(* IEC 61131-3 sources: Caravan/Archiv/12-04-19/Stations/MachineControl/MachineControl/Class/DayNightSplitter_Class, 1 file *)

(* ---- DayNightSplitter_Class.st ---- *)
(*!
<Class
	Name               = "DayNightSplitter_Class"
	Revision           = "0.0"
	RealtimeTask       = "false"
	CyclicTask         = "true"
	DefCyclictime      = "200 µs"
	BackgroundTask     = "false"
	Sigmatek           = "false"
	OSInterface        = "false"
	HighPriority       = "false"
	Automatic          = "false"
	UpdateMode         = "Prescan"
	SharedCommandTable = "true"
	Objectsize         = "(750,120)">
	<Channels>
		<Server Name="ClassSvr" Visualized="false" Initialize="false" WriteProtected="true" Retentive="false"/>
		<Server Name="DayFanMode" Visualized="true" Initialize="false" WriteProtected="false" Retentive="SRam"/>
		<Server Name="DayFanSpeed" Visualized="true" Initialize="false" WriteProtected="false" Retentive="SRam"/>
		<Server Name="DayHeaterON" Visualized="true" Initialize="false" WriteProtected="false" Retentive="SRam"/>
		<Server Name="DaySetRoomTemp" Visualized="true" Initialize="false" WriteProtected="false" Retentive="SRam"/>
		<Server Name="DaySetTempHZS" Visualized="true" Initialize="false" WriteProtected="false" Retentive="SRam"/>
		<Server Name="NightFanMode" Visualized="true" Initialize="false" WriteProtected="false" Retentive="SRam"/>
		<Server Name="NightFanSpeed" Visualized="true" Initialize="false" WriteProtected="false" Retentive="SRam"/>
		<Server Name="NightHeaterOn" Visualized="true" Initialize="false" WriteProtected="false" Retentive="SRam"/>
		<Server Name="NightSetRoomTemp" Visualized="true" Initialize="false" WriteProtected="false" Retentive="SRam"/>
		<Server Name="NightSetTempHZS" Visualized="true" Initialize="false" WriteProtected="false" Retentive="SRam"/>
		<Client Name="DesiredFanMode" Required="true" Internal="false"/>
		<Client Name="DesiredFanSpeed" Required="true" Internal="false"/>
		<Client Name="DesiredHeaterPWR" Required="true" Internal="false"/>
		<Client Name="DesiredHZSTemp" Required="true" Internal="false"/>
		<Client Name="DesiredRoomTemp" Required="true" Internal="false"/>
		<Client Name="OC_ToTimerClass" Required="true" Internal="false"/>
	</Channels>
</Class>
*)
DayNightSplitter_Class : CLASS
  //Servers:
	ClassSvr 	: SvrChCmd_DINT;
	DaySetTempHZS 	: SvrCh_DINT;
	DaySetRoomTemp 	: SvrCh_DINT;
	DayHeaterON 	: SvrCh_DINT;
	DayFanMode 	: SvrCh_DINT;
	DayFanSpeed 	: SvrCh_DINT;
	NightSetTempHZS 	: SvrCh_DINT;
	NightSetRoomTemp 	: SvrCh_DINT;
	NightHeaterOn 	: SvrCh_DINT;
	NightFanMode 	: SvrCh_DINT;
	NightFanSpeed 	: SvrCh_DINT;
  //Clients:
	OC_ToTimerClass 	: CltChCmd_Timer_Class;
	DesiredHZSTemp 	: CltCh_DINT;
	DesiredRoomTemp 	: CltCh_DINT;
	DesiredHeaterPWR 	: CltCh_DINT;
	DesiredFanMode 	: CltCh_DINT;
	DesiredFanSpeed 	: CltCh_DINT;
  //Variables:
  //Functions:

	FUNCTION VIRTUAL GLOBAL CyWork
		VAR_INPUT
			EAX 	: UDINT;
		END_VAR
		VAR_OUTPUT
			state (EAX) 	: UDINT;
		END_VAR;
  //Tables:
	FUNCTION @STD
		VAR_OUTPUT
			ret_code	: CONFSTATES;
		END_VAR;
	FUNCTION GLOBAL TAB @CT_;
END_CLASS;

#pragma usingLtd Timer_Class

FUNCTION VIRTUAL GLOBAL DayNightSplitter_Class::CyWork
	VAR_INPUT
		EAX 	: UDINT;
	END_VAR
	VAR_OUTPUT
		state (EAX) 	: UDINT;
	END_VAR

	state := READY;

END_FUNCTION
